{attribute 'GeneratedUsingTerminal: EL7041-0052-0016'}
{attribute addProperty BoxType "EL7041-0052-0016"}
{attribute addProperty Id "ENC_Status_compactAT %I*ENC_Status_compact_3C6E2C4411STM_StatusAT %I*STM_Status_36ED096F11ENC_Control_compactAT %Q*ENC_Control_compact_2E82BC435STM_ControlAT %Q*STM_Control_5A8B50163STM_VelocityAT %Q*STM_Velocity_A47A3F412WcStateAT %I*WcState_9091E0EB2InfoDataAT %I*InfoData_3B4F4E8A4"}
{attribute addProperty CRC "833429129"}
{attribute addProperty Size "38"}
TYPE EL7041_31AD1E89 EXTENDS EtcSlaveTerminalBase_947E5A46 :
STRUCT
	{attribute addProperty Name "ENC_Status_compact"}
	ENC_Status_compact : ENC_Status_compact_3C6E2C44;
	{attribute addProperty Name "STM_Status"}
	STM_Status : STM_Status_36ED096F;
	{attribute addProperty Name "ENC_Control_compact"}
	ENC_Control_compact : ENC_Control_compact_2E82BC43;
	{attribute addProperty Name "STM_Control"}
	STM_Control : STM_Control_5A8B5016;
	{attribute addProperty Name "STM_Velocity"}
	STM_Velocity : STM_Velocity_A47A3F41;
	{attribute addProperty Name "WcState"}
	WcState : WcState_9091E0EB;
	{attribute addProperty Name "InfoData"}
	InfoData : InfoData_3B4F4E8A;
END_STRUCT
END_TYPE

(* stored: Version 1.2.0.0, ProductVersion 3.1.4024.9
   DUT EL7041_31AD1E89: Id {5475ddbc-99b0-40c6-a148-9f82ee0b651a} *)
